{attribute 'qualified_only'}
VAR_GLOBAL
	InStream AT %MD0: InStream;
	OutStream AT %MD21: OutStream;
END_VAR

(* stored: Version 1.1.0.1, ProductVersion 3.1.4024.4
   GVL Streams: Id {35a4eca8-cff5-4d79-a04f-8802f49464c0} *)
